{attribute 'GeneratedUsingTerminal: EL2502-0010-0020'}
{attribute addProperty BoxType "EL2502-0010-0020"}
{attribute addProperty Id "SysTimeAT %I*ULINT8"}
{attribute addProperty CRC "282880325"}
{attribute addProperty Size "8"}
TYPE PWM_SysTime_Channel_10DC6945 EXTENDS InputBase_8311D824 :
STRUCT
	{attribute addProperty Name "SysTime"}
	SysTime AT %I* : ULINT;
END_STRUCT
END_TYPE

(* stored: Version 1.2.0.0, ProductVersion 3.1.4024.9
   DUT PWM_SysTime_Channel_10DC6945: Id {4af8e5c0-b449-4852-a6fc-172901ff794a} *)
